{attribute 'Tc2GvlVarNames'}
{attribute 'strict'}
TYPE e_TipoMacchinaTrasporti :
(
	Macchina_ZonaPal := 0,//Zona Pallettizzatore
	Macchina_ZonaBS := 1 //Zona BAnco Scelta
);
END_TYPE

(* stored: Version 1.1.0.1, ProductVersion 3.1.4024.11
   DUT e_TipoMacchinaTrasporti: Id {74390a1c-2d23-40cc-8e07-de882fa4ae81} *)
